# EPICS StreamDevice protocol: EPICS/Db/tdk.proto
# Author: Philip Weigel

Terminator = CR;

set_voltage {
	out "PV %f";
	in "OK";
}

set_current {
	out "PC %f";
	in "OK";
}

read_voltage {
	out "MV?";
	in "%f";
}

read_current {
	out "MC?";
	in "%f";
}

set_status {
	out "OUT %d";
	in "OK";
}

start {
	out "ADR 6";
	in "OK";
}

get_status {
	out "OUT?";
	in "%{OFF|ON}";

	@init {
		start;
	}
}
